PROGRAM MAIN
VAR	
	PosDegree AT %I*	: REAL	:= 0;
	PosPiston AT %I*	: REAL	:= 0;
	velocity AT %Q*		: REAL	:= 0;
END_VAR

END_PROGRAM

(* stored: Version 1.1.0.1, ProductVersion 3.1.4024.10
   POU MAIN: Id {05518f30-63f5-43e5-a500-2e4c842868d1}, SpecialFunc None *)
